TYPE "Type_FeedbackParam"
VERSION : 0.1
   STRUCT
      intval : Array[0.."MAX_FEEDBACKINT"] of Int := [5(-1)];
      dintval : Array[0.."MAX_FEEDBACKDINT"] of DInt := [48, 32000];
      realvalcfg : Array[0.."MAX_FEEDBACKREAL"] of Real;
      realval : Array[0.."MAX_FEEDBACKREAL"] of Real;
   END_STRUCT;

END_TYPE

